// TIA Portal V16 export
// export: Created 2022-11-17T15:49:29.9822396Z, ExportSetting WithDefaults, DisplayName Totally Integrated Automation Portal, DisplayVersion V16 Update 6, DisplayName TIA Portal Version Control Interface, DisplayVersion V16 Update 2, DisplayName TIA Portal Openness, DisplayVersion V16 Update 6, DisplayName SINAMICS Startdrive Advanced, DisplayVersion V16 Update 5, DisplayName SINAMICS Startdrive G130, G150, S120, S150, SINAMICS MV, S210, DisplayVersion V16 Update 5, DisplayName SINAMICS Startdrive G110M, G120, G120C, G120D, G120P, G115D, DisplayVersion V16 Update 5, DisplayName STEP 7 Professional, DisplayVersion V16 Update 6, DisplayName STEP 7 Safety, DisplayVersion V16, DisplayName WinCC Advanced, DisplayVersion V16 Update 6
FUNCTION "FC86_Conveyor_5_IN_3_OUT" : Void   // FC86, LAD
TITLE = Conveyor_5_IN_3_OUT
{ S7_Optimized_Access := 'TRUE' }
VERSION : 0.1
// 5+3 (Fitembal)
// stored: AutoNumber false, IsIECCheckEnabled false, SetENOAutomatically false, UDAEnableTagReadback false
   VAR_TEMP   // added for the SCL form of the ladder/FBD networks
      _w1 : Bool;
      _w2 : Bool;
   END_VAR
BEGIN

REGION Network 1: Manual operation for conveyor
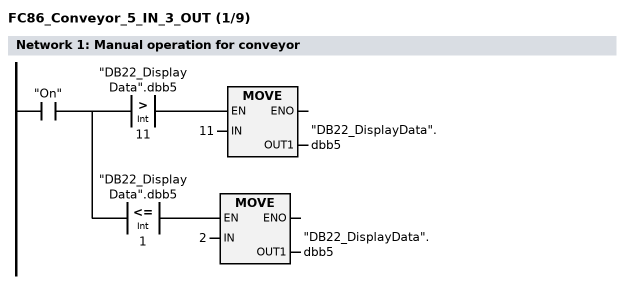
   RUNG wire#powerrail
      Contact( "On" )
      wire#w1
      { S7_Templates := "SrcType := Int" } GT_Contact(in1 := "DB22_DisplayData".dbb5, in2 := 11)
      { S7_GenerateENO := "TRUE" } Move(in := 11, out1 => "DB22_DisplayData".dbb5)
   END_RUNG
   RUNG wire#w1
      { S7_Templates := "SrcType := Int" } LE_Contact(in1 := "DB22_DisplayData".dbb5, in2 := 1)
      { S7_GenerateENO := "TRUE" } Move(in := 2, out1 => "DB22_DisplayData".dbb5)
   END_RUNG
   // the same network as SCL:
   IF "On" AND ("DB22_DisplayData".dbb5 > 11) THEN "DB22_DisplayData".dbb5 := 11; END_IF;
   IF "On" AND ("DB22_DisplayData".dbb5 <= 1) THEN "DB22_DisplayData".dbb5 := 2; END_IF;
END_REGION

REGION Network 2: Manual operation for conveyor
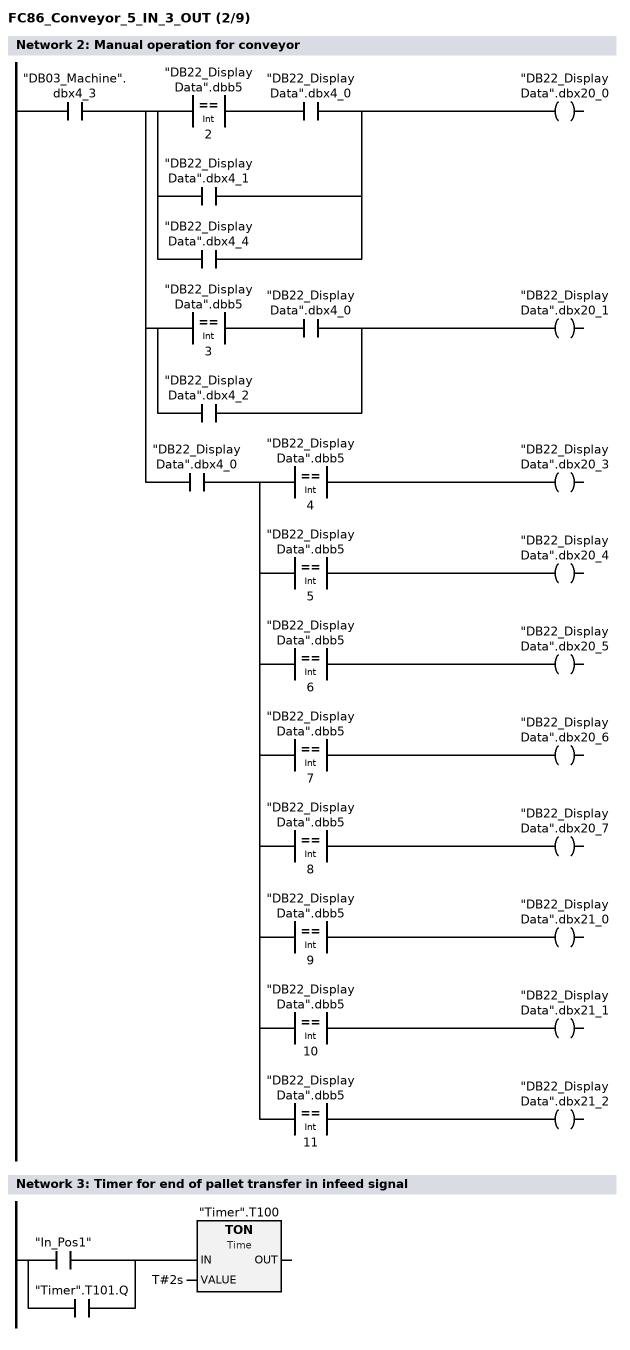
   RUNG wire#powerrail
      Contact( "DB03_Machine".dbx4_3 )
      wire#w1
      { S7_Templates := "SrcType := Int" } EQ_Contact(in1 := "DB22_DisplayData".dbb5, in2 := 2)
      Contact( "DB22_DisplayData".dbx4_0 )
      wire#w2
      Coil( "DB22_DisplayData".dbx20_0 )
   END_RUNG
   RUNG wire#w1
      Contact( "DB22_DisplayData".dbx4_1 )
   END_RUNG wire#w2
   RUNG wire#w1
      Contact( "DB22_DisplayData".dbx4_4 )
   END_RUNG wire#w2
   RUNG wire#w1
      { S7_Templates := "SrcType := Int" } EQ_Contact(in1 := "DB22_DisplayData".dbb5, in2 := 3)
      Contact( "DB22_DisplayData".dbx4_0 )
      wire#w3
      Coil( "DB22_DisplayData".dbx20_1 )
   END_RUNG
   RUNG wire#w1
      Contact( "DB22_DisplayData".dbx4_2 )
   END_RUNG wire#w3
   RUNG wire#w1
      Contact( "DB22_DisplayData".dbx4_0 )
      wire#w4
      { S7_Templates := "SrcType := Int" } EQ_Contact(in1 := "DB22_DisplayData".dbb5, in2 := 4)
      Coil( "DB22_DisplayData".dbx20_3 )
   END_RUNG
   RUNG wire#w4
      { S7_Templates := "SrcType := Int" } EQ_Contact(in1 := "DB22_DisplayData".dbb5, in2 := 5)
      Coil( "DB22_DisplayData".dbx20_4 )
   END_RUNG
   RUNG wire#w4
      { S7_Templates := "SrcType := Int" } EQ_Contact(in1 := "DB22_DisplayData".dbb5, in2 := 6)
      Coil( "DB22_DisplayData".dbx20_5 )
   END_RUNG
   RUNG wire#w4
      { S7_Templates := "SrcType := Int" } EQ_Contact(in1 := "DB22_DisplayData".dbb5, in2 := 7)
      Coil( "DB22_DisplayData".dbx20_6 )
   END_RUNG
   RUNG wire#w4
      { S7_Templates := "SrcType := Int" } EQ_Contact(in1 := "DB22_DisplayData".dbb5, in2 := 8)
      Coil( "DB22_DisplayData".dbx20_7 )
   END_RUNG
   RUNG wire#w4
      { S7_Templates := "SrcType := Int" } EQ_Contact(in1 := "DB22_DisplayData".dbb5, in2 := 9)
      Coil( "DB22_DisplayData".dbx21_0 )
   END_RUNG
   RUNG wire#w4
      { S7_Templates := "SrcType := Int" } EQ_Contact(in1 := "DB22_DisplayData".dbb5, in2 := 10)
      Coil( "DB22_DisplayData".dbx21_1 )
   END_RUNG
   RUNG wire#w4
      { S7_Templates := "SrcType := Int" } EQ_Contact(in1 := "DB22_DisplayData".dbb5, in2 := 11)
      Coil( "DB22_DisplayData".dbx21_2 )
   END_RUNG
   // the same network as SCL:
   "DB22_DisplayData".dbx20_0 := "DB03_Machine".dbx4_3 AND ((("DB22_DisplayData".dbb5 = 2) AND "DB22_DisplayData".dbx4_0) OR "DB22_DisplayData".dbx4_1 OR "DB22_DisplayData".dbx4_4);
   "DB22_DisplayData".dbx20_1 := "DB03_Machine".dbx4_3 AND ((("DB22_DisplayData".dbb5 = 3) AND "DB22_DisplayData".dbx4_0) OR "DB22_DisplayData".dbx4_2);
   #_w1 := "DB03_Machine".dbx4_3 AND "DB22_DisplayData".dbx4_0;
   "DB22_DisplayData".dbx20_3 := #_w1 AND ("DB22_DisplayData".dbb5 = 4);
   "DB22_DisplayData".dbx20_4 := #_w1 AND ("DB22_DisplayData".dbb5 = 5);
   "DB22_DisplayData".dbx20_5 := #_w1 AND ("DB22_DisplayData".dbb5 = 6);
   "DB22_DisplayData".dbx20_6 := #_w1 AND ("DB22_DisplayData".dbb5 = 7);
   "DB22_DisplayData".dbx20_7 := #_w1 AND ("DB22_DisplayData".dbb5 = 8);
   "DB22_DisplayData".dbx21_0 := #_w1 AND ("DB22_DisplayData".dbb5 = 9);
   "DB22_DisplayData".dbx21_1 := #_w1 AND ("DB22_DisplayData".dbb5 = 10);
   "DB22_DisplayData".dbx21_2 := #_w1 AND ("DB22_DisplayData".dbb5 = 11);
END_REGION

REGION Network 3: Timer for end of pallet transfer in infeed signal
   "Timer".T100.TON(IN := "In_Pos1" OR "Timer".T101.Q, PT := T#2s);   // TON coil
END_REGION

REGION Network 4: Timeout for conveyor pos1
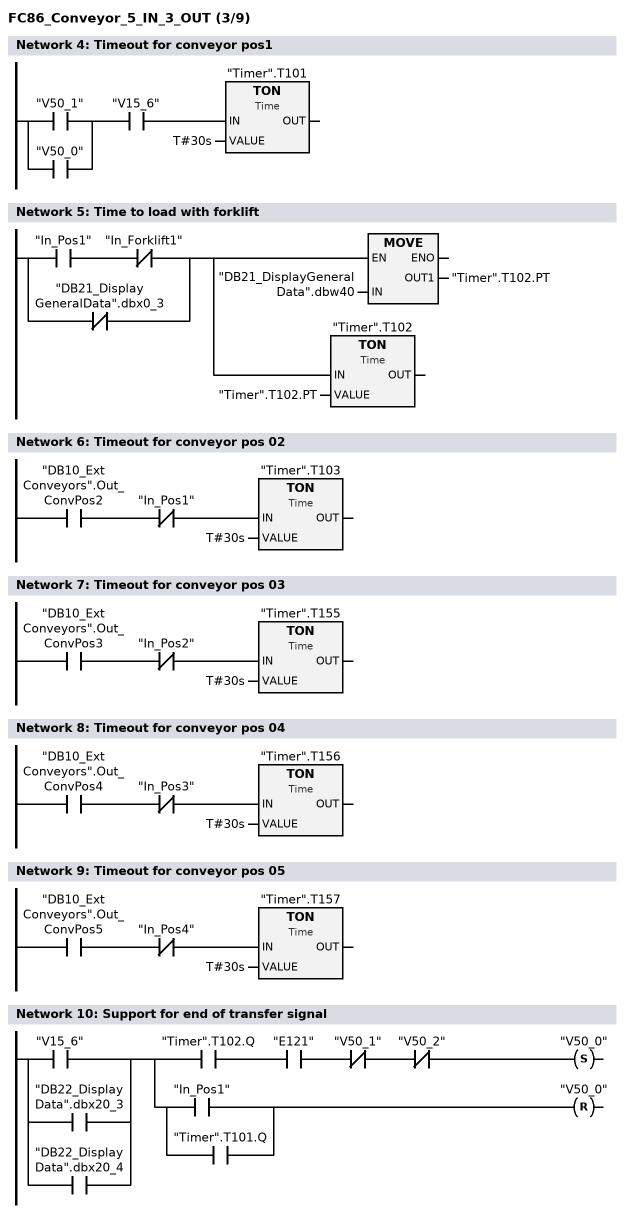
   "Timer".T101.TON(IN := ("V50_1" OR "V50_0") AND "V15_6", PT := T#30s);   // TON coil
END_REGION

REGION Network 5: Time to load with forklift
   #_w1 := ("In_Pos1" AND NOT "In_Forklift1") OR NOT "DB21_DisplayGeneralData".dbx0_3;
   IF #_w1 THEN "Timer".T102.PT := "DB21_DisplayGeneralData".dbw40; END_IF;
   "Timer".T102.TON(IN := #_w1, PT := "Timer".T102.PT);   // TON coil
END_REGION

REGION Network 6: Timeout for conveyor pos 02
   "Timer".T103.TON(IN := "DB10_ExtConveyors".Out_ConvPos2 AND NOT "In_Pos1", PT := T#30s);   // TON coil
END_REGION

REGION Network 7: Timeout for conveyor pos 03
   "Timer".T155.TON(IN := "DB10_ExtConveyors".Out_ConvPos3 AND NOT "In_Pos2", PT := T#30s);   // TON coil
END_REGION

REGION Network 8: Timeout for conveyor pos 04
   "Timer".T156.TON(IN := "DB10_ExtConveyors".Out_ConvPos4 AND NOT "In_Pos3", PT := T#30s);   // TON coil
END_REGION

REGION Network 9: Timeout for conveyor pos 05
   "Timer".T157.TON(IN := "DB10_ExtConveyors".Out_ConvPos5 AND NOT "In_Pos4", PT := T#30s);   // TON coil
END_REGION

REGION Network 10: Support for end of transfer signal
   RUNG wire#powerrail
      Contact( "V15_6" )
      wire#w1
      Contact( "Timer".T102.Q )
      Contact( "E121" )
      I_Contact( "V50_1" )
      I_Contact( "V50_2" )
      S_Coil( "V50_0" )
   END_RUNG
   RUNG wire#powerrail
      Contact( "DB22_DisplayData".dbx20_3 )
   END_RUNG wire#w1
   RUNG wire#powerrail
      Contact( "DB22_DisplayData".dbx20_4 )
   END_RUNG wire#w1
   RUNG wire#w1
      Contact( "In_Pos1" )
      wire#w2
      R_Coil( "V50_0" )
   END_RUNG
   RUNG wire#w1
      Contact( "Timer".T101.Q )
   END_RUNG wire#w2
   // the same network as SCL:
   #_w1 := "V15_6" OR "DB22_DisplayData".dbx20_3 OR "DB22_DisplayData".dbx20_4;
   IF #_w1 AND "Timer".T102.Q AND "E121" AND NOT "V50_1" AND NOT "V50_2" THEN "V50_0" := TRUE; END_IF;
   IF #_w1 AND ("In_Pos1" OR "Timer".T101.Q) THEN "V50_0" := FALSE; END_IF;
END_REGION

REGION Network 11: Transit memory for conveyor pos1
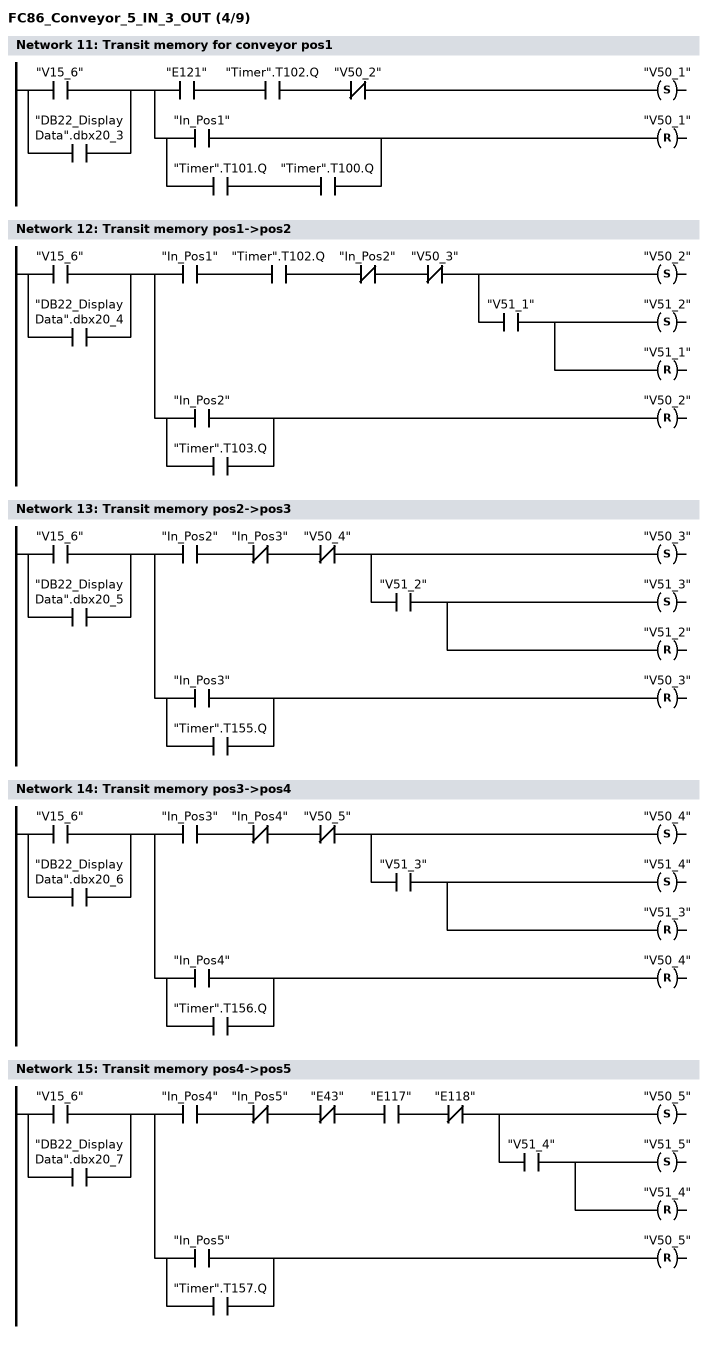
   RUNG wire#powerrail
      Contact( "V15_6" )
      wire#w1
      Contact( "E121" )
      Contact( "Timer".T102.Q )
      I_Contact( "V50_2" )
      S_Coil( "V50_1" )
   END_RUNG
   RUNG wire#powerrail
      Contact( "DB22_DisplayData".dbx20_3 )
   END_RUNG wire#w1
   RUNG wire#w1
      Contact( "In_Pos1" )
      wire#w2
      R_Coil( "V50_1" )
   END_RUNG
   RUNG wire#w1
      Contact( "Timer".T101.Q )
      Contact( "Timer".T100.Q )
   END_RUNG wire#w2
   // the same network as SCL:
   #_w1 := "V15_6" OR "DB22_DisplayData".dbx20_3;
   IF #_w1 AND "E121" AND "Timer".T102.Q AND NOT "V50_2" THEN "V50_1" := TRUE; END_IF;
   IF #_w1 AND ("In_Pos1" OR ("Timer".T101.Q AND "Timer".T100.Q)) THEN "V50_1" := FALSE; END_IF;
END_REGION

REGION Network 12: Transit memory pos1->pos2
   RUNG wire#powerrail
      Contact( "V15_6" )
      wire#w1
      Contact( "In_Pos1" )
      Contact( "Timer".T102.Q )
      I_Contact( "In_Pos2" )
      I_Contact( "V50_3" )
      wire#w2
      S_Coil( "V50_2" )
   END_RUNG
   RUNG wire#powerrail
      Contact( "DB22_DisplayData".dbx20_4 )
   END_RUNG wire#w1
   RUNG wire#w2
      Contact( "V51_1" )
      wire#w3
      S_Coil( "V51_2" )
   END_RUNG
   RUNG wire#w3
      R_Coil( "V51_1" )
   END_RUNG
   RUNG wire#w1
      Contact( "In_Pos2" )
      wire#w4
      R_Coil( "V50_2" )
   END_RUNG
   RUNG wire#w1
      Contact( "Timer".T103.Q )
   END_RUNG wire#w4
   // the same network as SCL:
   #_w1 := "V15_6" OR "DB22_DisplayData".dbx20_4;
   #_w2 := #_w1 AND "In_Pos1" AND "Timer".T102.Q AND NOT "In_Pos2" AND NOT "V50_3";
   IF #_w2 THEN "V50_2" := TRUE; END_IF;
   IF #_w2 AND "V51_1" THEN
       "V51_2" := TRUE;
       "V51_1" := FALSE;
   END_IF;
   IF #_w1 AND ("In_Pos2" OR "Timer".T103.Q) THEN "V50_2" := FALSE; END_IF;
END_REGION

REGION Network 13: Transit memory pos2->pos3
   RUNG wire#powerrail
      Contact( "V15_6" )
      wire#w1
      Contact( "In_Pos2" )
      I_Contact( "In_Pos3" )
      I_Contact( "V50_4" )
      wire#w2
      S_Coil( "V50_3" )
   END_RUNG
   RUNG wire#powerrail
      Contact( "DB22_DisplayData".dbx20_5 )
   END_RUNG wire#w1
   RUNG wire#w2
      Contact( "V51_2" )
      wire#w3
      S_Coil( "V51_3" )
   END_RUNG
   RUNG wire#w3
      R_Coil( "V51_2" )
   END_RUNG
   RUNG wire#w1
      Contact( "In_Pos3" )
      wire#w4
      R_Coil( "V50_3" )
   END_RUNG
   RUNG wire#w1
      Contact( "Timer".T155.Q )
   END_RUNG wire#w4
   // the same network as SCL:
   #_w1 := "V15_6" OR "DB22_DisplayData".dbx20_5;
   #_w2 := #_w1 AND "In_Pos2" AND NOT "In_Pos3" AND NOT "V50_4";
   IF #_w2 THEN "V50_3" := TRUE; END_IF;
   IF #_w2 AND "V51_2" THEN
       "V51_3" := TRUE;
       "V51_2" := FALSE;
   END_IF;
   IF #_w1 AND ("In_Pos3" OR "Timer".T155.Q) THEN "V50_3" := FALSE; END_IF;
END_REGION

REGION Network 14: Transit memory pos3->pos4
   RUNG wire#powerrail
      Contact( "V15_6" )
      wire#w1
      Contact( "In_Pos3" )
      I_Contact( "In_Pos4" )
      I_Contact( "V50_5" )
      wire#w2
      S_Coil( "V50_4" )
   END_RUNG
   RUNG wire#powerrail
      Contact( "DB22_DisplayData".dbx20_6 )
   END_RUNG wire#w1
   RUNG wire#w2
      Contact( "V51_3" )
      wire#w3
      S_Coil( "V51_4" )
   END_RUNG
   RUNG wire#w3
      R_Coil( "V51_3" )
   END_RUNG
   RUNG wire#w1
      Contact( "In_Pos4" )
      wire#w4
      R_Coil( "V50_4" )
   END_RUNG
   RUNG wire#w1
      Contact( "Timer".T156.Q )
   END_RUNG wire#w4
   // the same network as SCL:
   #_w1 := "V15_6" OR "DB22_DisplayData".dbx20_6;
   #_w2 := #_w1 AND "In_Pos3" AND NOT "In_Pos4" AND NOT "V50_5";
   IF #_w2 THEN "V50_4" := TRUE; END_IF;
   IF #_w2 AND "V51_3" THEN
       "V51_4" := TRUE;
       "V51_3" := FALSE;
   END_IF;
   IF #_w1 AND ("In_Pos4" OR "Timer".T156.Q) THEN "V50_4" := FALSE; END_IF;
END_REGION

REGION Network 15: Transit memory pos4->pos5
   RUNG wire#powerrail
      Contact( "V15_6" )
      wire#w1
      Contact( "In_Pos4" )
      I_Contact( "In_Pos5" )
      I_Contact( "E43" )
      Contact( "E117" )
      I_Contact( "E118" )
      wire#w2
      S_Coil( "V50_5" )
   END_RUNG
   RUNG wire#powerrail
      Contact( "DB22_DisplayData".dbx20_7 )
   END_RUNG wire#w1
   RUNG wire#w2
      Contact( "V51_4" )
      wire#w3
      S_Coil( "V51_5" )
   END_RUNG
   RUNG wire#w3
      R_Coil( "V51_4" )
   END_RUNG
   RUNG wire#w1
      Contact( "In_Pos5" )
      wire#w4
      R_Coil( "V50_5" )
   END_RUNG
   RUNG wire#w1
      Contact( "Timer".T157.Q )
   END_RUNG wire#w4
   // the same network as SCL:
   #_w1 := "V15_6" OR "DB22_DisplayData".dbx20_7;
   #_w2 := #_w1 AND "In_Pos4" AND NOT "In_Pos5" AND NOT "E43" AND "E117" AND NOT "E118";
   IF #_w2 THEN "V50_5" := TRUE; END_IF;
   IF #_w2 AND "V51_4" THEN
       "V51_5" := TRUE;
       "V51_4" := FALSE;
   END_IF;
   IF #_w1 AND ("In_Pos5" OR "Timer".T157.Q) THEN "V50_5" := FALSE; END_IF;
END_REGION

REGION Network 16: Ready to receive pallet in infeed signal
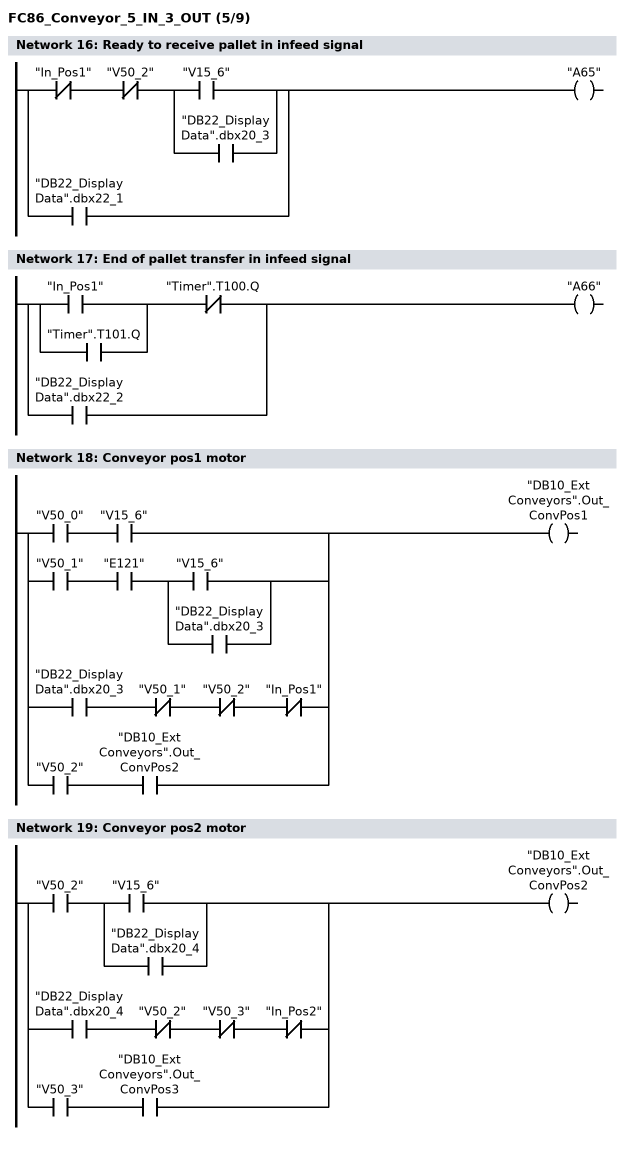
   RUNG wire#powerrail
      I_Contact( "In_Pos1" )
      I_Contact( "V50_2" )
      wire#w1
      Contact( "V15_6" )
      wire#w2
      Coil( "A65" )
   END_RUNG
   RUNG wire#w1
      Contact( "DB22_DisplayData".dbx20_3 )
   END_RUNG wire#w2
   RUNG wire#powerrail
      Contact( "DB22_DisplayData".dbx22_1 )
   END_RUNG wire#w2
   // the same network as SCL:
   "A65" := (NOT "In_Pos1" AND NOT "V50_2" AND ("V15_6" OR "DB22_DisplayData".dbx20_3)) OR "DB22_DisplayData".dbx22_1;
END_REGION

REGION Network 17: End of pallet transfer in infeed signal
   RUNG wire#powerrail
      Contact( "In_Pos1" )
      wire#w1
      I_Contact( "Timer".T100.Q )
      wire#w2
      Coil( "A66" )
   END_RUNG
   RUNG wire#powerrail
      Contact( "Timer".T101.Q )
   END_RUNG wire#w1
   RUNG wire#powerrail
      Contact( "DB22_DisplayData".dbx22_2 )
   END_RUNG wire#w2
   // the same network as SCL:
   "A66" := (("In_Pos1" OR "Timer".T101.Q) AND NOT "Timer".T100.Q) OR "DB22_DisplayData".dbx22_2;
END_REGION

REGION Network 18: Conveyor pos1 motor
   RUNG wire#powerrail
      Contact( "V50_0" )
      Contact( "V15_6" )
      wire#w1
      Coil( "DB10_ExtConveyors".Out_ConvPos1 )
   END_RUNG
   RUNG wire#powerrail
      Contact( "V50_1" )
      Contact( "E121" )
      wire#w2
      Contact( "V15_6" )
   END_RUNG wire#w1
   RUNG wire#w2
      Contact( "DB22_DisplayData".dbx20_3 )
   END_RUNG wire#w1
   RUNG wire#powerrail
      Contact( "DB22_DisplayData".dbx20_3 )
      I_Contact( "V50_1" )
      I_Contact( "V50_2" )
      I_Contact( "In_Pos1" )
   END_RUNG wire#w1
   RUNG wire#powerrail
      Contact( "V50_2" )
      Contact( "DB10_ExtConveyors".Out_ConvPos2 )
   END_RUNG wire#w1
   // the same network as SCL:
   "DB10_ExtConveyors".Out_ConvPos1 := ("V50_0" AND "V15_6") OR ("V50_1" AND "E121" AND ("V15_6" OR "DB22_DisplayData".dbx20_3)) OR ("DB22_DisplayData".dbx20_3 AND NOT "V50_1" AND NOT "V50_2" AND NOT "In_Pos1") OR ("V50_2" AND "DB10_ExtConveyors".Out_ConvPos2);
END_REGION

REGION Network 19: Conveyor pos2 motor
   RUNG wire#powerrail
      Contact( "V50_2" )
      wire#w1
      Contact( "V15_6" )
      wire#w2
      Coil( "DB10_ExtConveyors".Out_ConvPos2 )
   END_RUNG
   RUNG wire#w1
      Contact( "DB22_DisplayData".dbx20_4 )
   END_RUNG wire#w2
   RUNG wire#powerrail
      Contact( "DB22_DisplayData".dbx20_4 )
      I_Contact( "V50_2" )
      I_Contact( "V50_3" )
      I_Contact( "In_Pos2" )
   END_RUNG wire#w2
   RUNG wire#powerrail
      Contact( "V50_3" )
      Contact( "DB10_ExtConveyors".Out_ConvPos3 )
   END_RUNG wire#w2
   // the same network as SCL:
   "DB10_ExtConveyors".Out_ConvPos2 := ("V50_2" AND ("V15_6" OR "DB22_DisplayData".dbx20_4)) OR ("DB22_DisplayData".dbx20_4 AND NOT "V50_2" AND NOT "V50_3" AND NOT "In_Pos2") OR ("V50_3" AND "DB10_ExtConveyors".Out_ConvPos3);
END_REGION

REGION Network 20: Conveyor pos3 motor
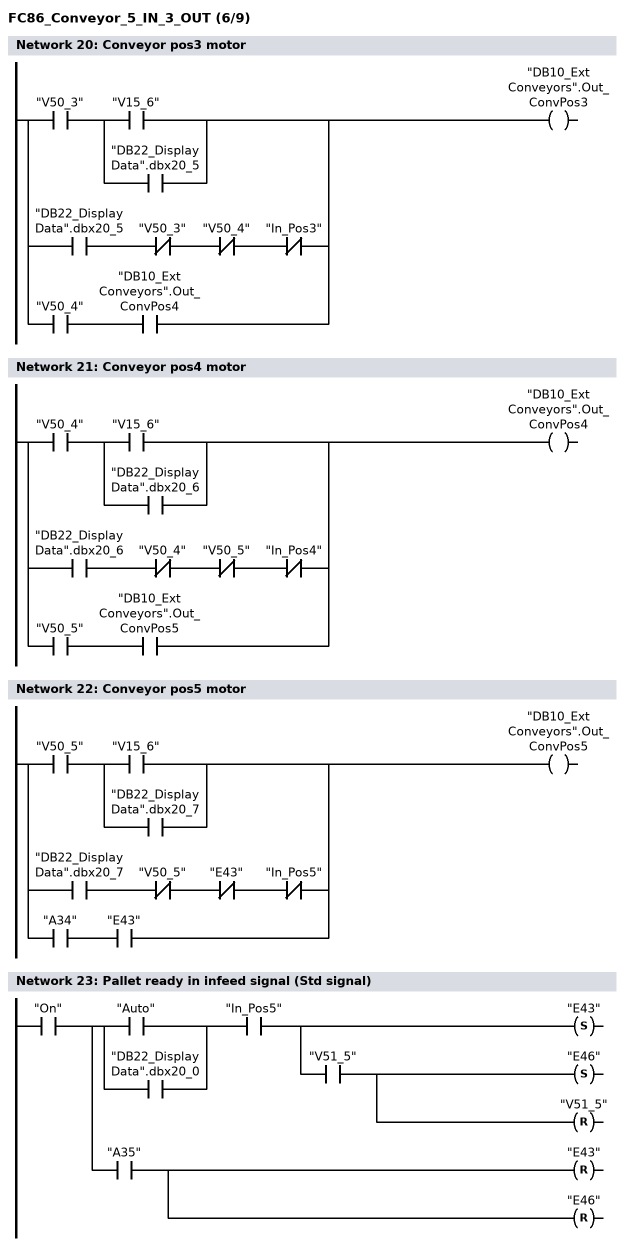
   RUNG wire#powerrail
      Contact( "V50_3" )
      wire#w1
      Contact( "V15_6" )
      wire#w2
      Coil( "DB10_ExtConveyors".Out_ConvPos3 )
   END_RUNG
   RUNG wire#w1
      Contact( "DB22_DisplayData".dbx20_5 )
   END_RUNG wire#w2
   RUNG wire#powerrail
      Contact( "DB22_DisplayData".dbx20_5 )
      I_Contact( "V50_3" )
      I_Contact( "V50_4" )
      I_Contact( "In_Pos3" )
   END_RUNG wire#w2
   RUNG wire#powerrail
      Contact( "V50_4" )
      Contact( "DB10_ExtConveyors".Out_ConvPos4 )
   END_RUNG wire#w2
   // the same network as SCL:
   "DB10_ExtConveyors".Out_ConvPos3 := ("V50_3" AND ("V15_6" OR "DB22_DisplayData".dbx20_5)) OR ("DB22_DisplayData".dbx20_5 AND NOT "V50_3" AND NOT "V50_4" AND NOT "In_Pos3") OR ("V50_4" AND "DB10_ExtConveyors".Out_ConvPos4);
END_REGION

REGION Network 21: Conveyor pos4 motor
   RUNG wire#powerrail
      Contact( "V50_4" )
      wire#w1
      Contact( "V15_6" )
      wire#w2
      Coil( "DB10_ExtConveyors".Out_ConvPos4 )
   END_RUNG
   RUNG wire#w1
      Contact( "DB22_DisplayData".dbx20_6 )
   END_RUNG wire#w2
   RUNG wire#powerrail
      Contact( "DB22_DisplayData".dbx20_6 )
      I_Contact( "V50_4" )
      I_Contact( "V50_5" )
      I_Contact( "In_Pos4" )
   END_RUNG wire#w2
   RUNG wire#powerrail
      Contact( "V50_5" )
      Contact( "DB10_ExtConveyors".Out_ConvPos5 )
   END_RUNG wire#w2
   // the same network as SCL:
   "DB10_ExtConveyors".Out_ConvPos4 := ("V50_4" AND ("V15_6" OR "DB22_DisplayData".dbx20_6)) OR ("DB22_DisplayData".dbx20_6 AND NOT "V50_4" AND NOT "V50_5" AND NOT "In_Pos4") OR ("V50_5" AND "DB10_ExtConveyors".Out_ConvPos5);
END_REGION

REGION Network 22: Conveyor pos5 motor
   RUNG wire#powerrail
      Contact( "V50_5" )
      wire#w1
      Contact( "V15_6" )
      wire#w2
      Coil( "DB10_ExtConveyors".Out_ConvPos5 )
   END_RUNG
   RUNG wire#w1
      Contact( "DB22_DisplayData".dbx20_7 )
   END_RUNG wire#w2
   RUNG wire#powerrail
      Contact( "DB22_DisplayData".dbx20_7 )
      I_Contact( "V50_5" )
      I_Contact( "E43" )
      I_Contact( "In_Pos5" )
   END_RUNG wire#w2
   RUNG wire#powerrail
      Contact( "A34" )
      Contact( "E43" )
   END_RUNG wire#w2
   // the same network as SCL:
   "DB10_ExtConveyors".Out_ConvPos5 := ("V50_5" AND ("V15_6" OR "DB22_DisplayData".dbx20_7)) OR ("DB22_DisplayData".dbx20_7 AND NOT "V50_5" AND NOT "E43" AND NOT "In_Pos5") OR ("A34" AND "E43");
END_REGION

REGION Network 23: Pallet ready in infeed signal (Std signal)
   RUNG wire#powerrail
      Contact( "On" )
      wire#w1
      Contact( "Auto" )
      wire#w2
      Contact( "In_Pos5" )
      wire#w3
      S_Coil( "E43" )
   END_RUNG
   RUNG wire#w1
      Contact( "DB22_DisplayData".dbx20_0 )
   END_RUNG wire#w2
   RUNG wire#w3
      Contact( "V51_5" )
      wire#w4
      S_Coil( "E46" )
   END_RUNG
   RUNG wire#w4
      R_Coil( "V51_5" )
   END_RUNG
   RUNG wire#w1
      Contact( "A35" )
      wire#w5
      R_Coil( "E43" )
   END_RUNG
   RUNG wire#w5
      R_Coil( "E46" )
   END_RUNG
   // the same network as SCL:
   #_w1 := "On" AND ("Auto" OR "DB22_DisplayData".dbx20_0) AND "In_Pos5";
   IF #_w1 THEN "E43" := TRUE; END_IF;
   IF #_w1 AND "V51_5" THEN
       "E46" := TRUE;
       "V51_5" := FALSE;
   END_IF;
   IF "On" AND "A35" THEN
       "E43" := FALSE;
       "E46" := FALSE;
   END_IF;
END_REGION

REGION Network 24: Memory to exclude wrapping in pos 1
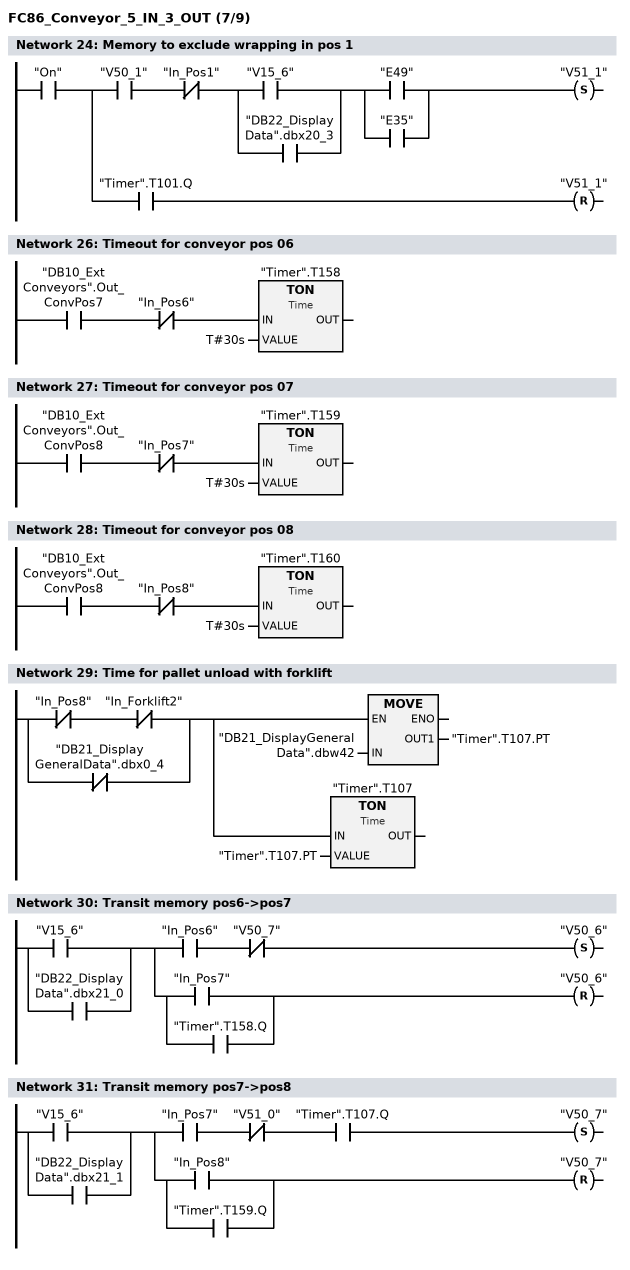
   RUNG wire#powerrail
      Contact( "On" )
      wire#w1
      Contact( "V50_1" )
      I_Contact( "In_Pos1" )
      wire#w2
      Contact( "V15_6" )
      wire#w3
      Contact( "E49" )
      wire#w4
      S_Coil( "V51_1" )
   END_RUNG
   RUNG wire#w2
      Contact( "DB22_DisplayData".dbx20_3 )
   END_RUNG wire#w3
   RUNG wire#w3
      Contact( "E35" )
   END_RUNG wire#w4
   RUNG wire#w1
      Contact( "Timer".T101.Q )
      R_Coil( "V51_1" )
   END_RUNG
   // the same network as SCL:
   IF "On" AND "V50_1" AND NOT "In_Pos1" AND ("V15_6" OR "DB22_DisplayData".dbx20_3) AND ("E49" OR "E35") THEN
       "V51_1" := TRUE;
   END_IF;
   IF "On" AND "Timer".T101.Q THEN "V51_1" := FALSE; END_IF;
END_REGION

REGION Network 25: >>>>>>> OUTFEED CONVEYOR <<<<<<<<
END_REGION

REGION Network 26: Timeout for conveyor pos 06
   "Timer".T158.TON(IN := "DB10_ExtConveyors".Out_ConvPos7 AND NOT "In_Pos6", PT := T#30s);   // TON coil
END_REGION

REGION Network 27: Timeout for conveyor pos 07
   "Timer".T159.TON(IN := "DB10_ExtConveyors".Out_ConvPos8 AND NOT "In_Pos7", PT := T#30s);   // TON coil
END_REGION

REGION Network 28: Timeout for conveyor pos 08
   "Timer".T160.TON(IN := "DB10_ExtConveyors".Out_ConvPos8 AND NOT "In_Pos8", PT := T#30s);   // TON coil
END_REGION

REGION Network 29: Time for pallet unload with forklift
   #_w1 := (NOT "In_Pos8" AND NOT "In_Forklift2") OR NOT "DB21_DisplayGeneralData".dbx0_4;
   IF #_w1 THEN "Timer".T107.PT := "DB21_DisplayGeneralData".dbw42; END_IF;
   "Timer".T107.TON(IN := #_w1, PT := "Timer".T107.PT);   // TON coil
END_REGION

REGION Network 30: Transit memory pos6->pos7
   RUNG wire#powerrail
      Contact( "V15_6" )
      wire#w1
      Contact( "In_Pos6" )
      I_Contact( "V50_7" )
      S_Coil( "V50_6" )
   END_RUNG
   RUNG wire#powerrail
      Contact( "DB22_DisplayData".dbx21_0 )
   END_RUNG wire#w1
   RUNG wire#w1
      Contact( "In_Pos7" )
      wire#w2
      R_Coil( "V50_6" )
   END_RUNG
   RUNG wire#w1
      Contact( "Timer".T158.Q )
   END_RUNG wire#w2
   // the same network as SCL:
   #_w1 := "V15_6" OR "DB22_DisplayData".dbx21_0;
   IF #_w1 AND "In_Pos6" AND NOT "V50_7" THEN "V50_6" := TRUE; END_IF;
   IF #_w1 AND ("In_Pos7" OR "Timer".T158.Q) THEN "V50_6" := FALSE; END_IF;
END_REGION

REGION Network 31: Transit memory pos7->pos8
   RUNG wire#powerrail
      Contact( "V15_6" )
      wire#w1
      Contact( "In_Pos7" )
      I_Contact( "V51_0" )
      Contact( "Timer".T107.Q )
      S_Coil( "V50_7" )
   END_RUNG
   RUNG wire#powerrail
      Contact( "DB22_DisplayData".dbx21_1 )
   END_RUNG wire#w1
   RUNG wire#w1
      Contact( "In_Pos8" )
      wire#w2
      R_Coil( "V50_7" )
   END_RUNG
   RUNG wire#w1
      Contact( "Timer".T159.Q )
   END_RUNG wire#w2
   // the same network as SCL:
   #_w1 := "V15_6" OR "DB22_DisplayData".dbx21_1;
   IF #_w1 AND "In_Pos7" AND NOT "V51_0" AND "Timer".T107.Q THEN "V50_7" := TRUE; END_IF;
   IF #_w1 AND ("In_Pos8" OR "Timer".T159.Q) THEN "V50_7" := FALSE; END_IF;
END_REGION

REGION Network 32: Outfeed conveyor pos.8 unload
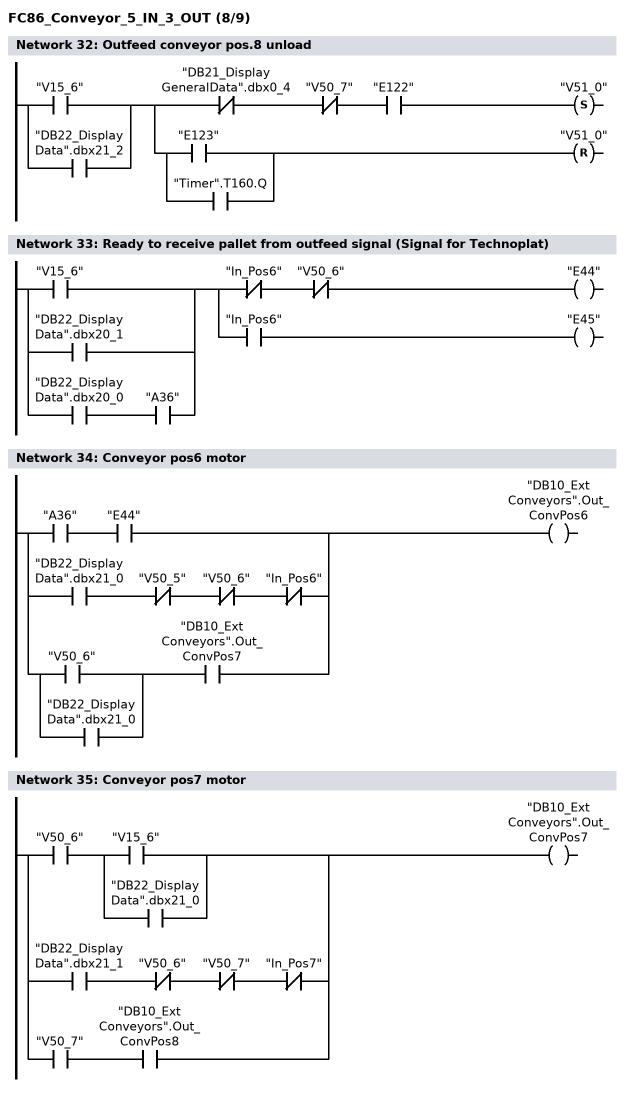
   RUNG wire#powerrail
      Contact( "V15_6" )
      wire#w1
      I_Contact( "DB21_DisplayGeneralData".dbx0_4 )
      I_Contact( "V50_7" )
      Contact( "E122" )
      S_Coil( "V51_0" )
   END_RUNG
   RUNG wire#powerrail
      Contact( "DB22_DisplayData".dbx21_2 )
   END_RUNG wire#w1
   RUNG wire#w1
      Contact( "E123" )
      wire#w2
      R_Coil( "V51_0" )
   END_RUNG
   RUNG wire#w1
      Contact( "Timer".T160.Q )
   END_RUNG wire#w2
   // the same network as SCL:
   #_w1 := "V15_6" OR "DB22_DisplayData".dbx21_2;
   IF #_w1 AND NOT "DB21_DisplayGeneralData".dbx0_4 AND NOT "V50_7" AND "E122" THEN "V51_0" := TRUE; END_IF;
   IF #_w1 AND ("E123" OR "Timer".T160.Q) THEN "V51_0" := FALSE; END_IF;
END_REGION

REGION Network 33: Ready to receive pallet from outfeed signal (Signal for Technoplat)
   RUNG wire#powerrail
      Contact( "V15_6" )
      wire#w1
      I_Contact( "In_Pos6" )
      I_Contact( "V50_6" )
      Coil( "E44" )
   END_RUNG
   RUNG wire#powerrail
      Contact( "DB22_DisplayData".dbx20_1 )
   END_RUNG wire#w1
   RUNG wire#powerrail
      Contact( "DB22_DisplayData".dbx20_0 )
      Contact( "A36" )
   END_RUNG wire#w1
   RUNG wire#w1
      Contact( "In_Pos6" )
      Coil( "E45" )
   END_RUNG
   // the same network as SCL:
   #_w1 := "V15_6" OR "DB22_DisplayData".dbx20_1 OR ("DB22_DisplayData".dbx20_0 AND "A36");
   "E44" := #_w1 AND NOT "In_Pos6" AND NOT "V50_6";
   "E45" := #_w1 AND "In_Pos6";
END_REGION

REGION Network 34: Conveyor pos6 motor
   RUNG wire#powerrail
      Contact( "A36" )
      Contact( "E44" )
      wire#w1
      Coil( "DB10_ExtConveyors".Out_ConvPos6 )
   END_RUNG
   RUNG wire#powerrail
      Contact( "DB22_DisplayData".dbx21_0 )
      I_Contact( "V50_5" )
      I_Contact( "V50_6" )
      I_Contact( "In_Pos6" )
   END_RUNG wire#w1
   RUNG wire#powerrail
      Contact( "V50_6" )
      wire#w2
      Contact( "DB10_ExtConveyors".Out_ConvPos7 )
   END_RUNG wire#w1
   RUNG wire#powerrail
      Contact( "DB22_DisplayData".dbx21_0 )
   END_RUNG wire#w2
   // the same network as SCL:
   "DB10_ExtConveyors".Out_ConvPos6 := ("A36" AND "E44") OR ("DB22_DisplayData".dbx21_0 AND NOT "V50_5" AND NOT "V50_6" AND NOT "In_Pos6") OR (("V50_6" OR "DB22_DisplayData".dbx21_0) AND "DB10_ExtConveyors".Out_ConvPos7);
END_REGION

REGION Network 35: Conveyor pos7 motor
   RUNG wire#powerrail
      Contact( "V50_6" )
      wire#w1
      Contact( "V15_6" )
      wire#w2
      Coil( "DB10_ExtConveyors".Out_ConvPos7 )
   END_RUNG
   RUNG wire#w1
      Contact( "DB22_DisplayData".dbx21_0 )
   END_RUNG wire#w2
   RUNG wire#powerrail
      Contact( "DB22_DisplayData".dbx21_1 )
      I_Contact( "V50_6" )
      I_Contact( "V50_7" )
      I_Contact( "In_Pos7" )
   END_RUNG wire#w2
   RUNG wire#powerrail
      Contact( "V50_7" )
      Contact( "DB10_ExtConveyors".Out_ConvPos8 )
   END_RUNG wire#w2
   // the same network as SCL:
   "DB10_ExtConveyors".Out_ConvPos7 := ("V50_6" AND ("V15_6" OR "DB22_DisplayData".dbx21_0)) OR ("DB22_DisplayData".dbx21_1 AND NOT "V50_6" AND NOT "V50_7" AND NOT "In_Pos7") OR ("V50_7" AND "DB10_ExtConveyors".Out_ConvPos8);
END_REGION

REGION Network 36: Conveyor pos8 motor
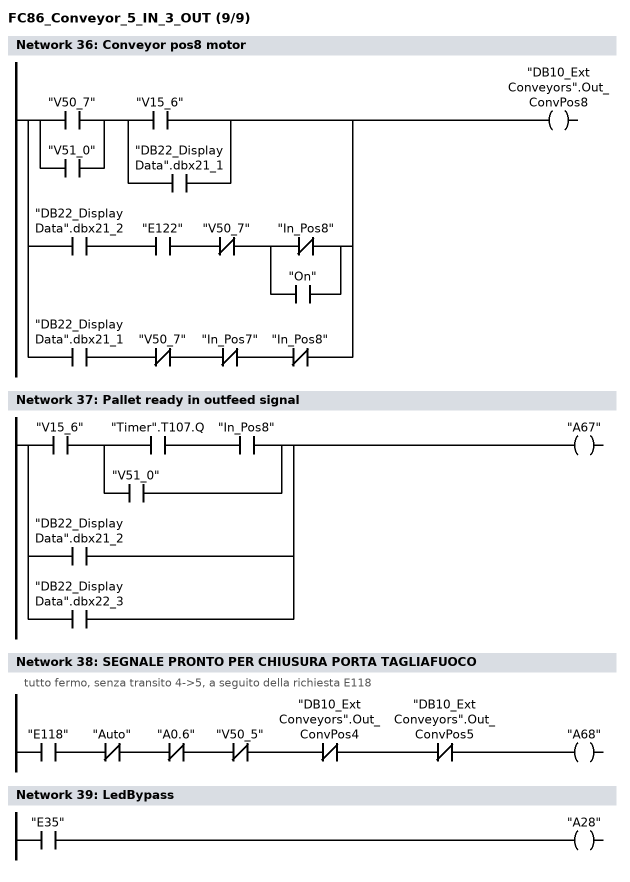
   RUNG wire#powerrail
      Contact( "V50_7" )
      wire#w1
      Contact( "V15_6" )
      wire#w2
      Coil( "DB10_ExtConveyors".Out_ConvPos8 )
   END_RUNG
   RUNG wire#powerrail
      Contact( "V51_0" )
   END_RUNG wire#w1
   RUNG wire#w1
      Contact( "DB22_DisplayData".dbx21_1 )
   END_RUNG wire#w2
   RUNG wire#powerrail
      Contact( "DB22_DisplayData".dbx21_2 )
      Contact( "E122" )
      I_Contact( "V50_7" )
      wire#w3
      I_Contact( "In_Pos8" )
   END_RUNG wire#w2
   RUNG wire#w3
      Contact( "On" )
   END_RUNG wire#w2
   RUNG wire#powerrail
      Contact( "DB22_DisplayData".dbx21_1 )
      I_Contact( "V50_7" )
      I_Contact( "In_Pos7" )
      I_Contact( "In_Pos8" )
   END_RUNG wire#w2
   // the same network as SCL:
   "DB10_ExtConveyors".Out_ConvPos8 := (("V50_7" OR "V51_0") AND ("V15_6" OR "DB22_DisplayData".dbx21_1)) OR ("DB22_DisplayData".dbx21_2 AND "E122" AND NOT "V50_7" AND (NOT "In_Pos8" OR "On")) OR ("DB22_DisplayData".dbx21_1 AND NOT "V50_7" AND NOT "In_Pos7" AND NOT "In_Pos8");
END_REGION

REGION Network 37: Pallet ready in outfeed signal
   RUNG wire#powerrail
      Contact( "V15_6" )
      wire#w1
      Contact( "Timer".T107.Q )
      Contact( "In_Pos8" )
      wire#w2
      Coil( "A67" )
   END_RUNG
   RUNG wire#w1
      Contact( "V51_0" )
   END_RUNG wire#w2
   RUNG wire#powerrail
      Contact( "DB22_DisplayData".dbx21_2 )
   END_RUNG wire#w2
   RUNG wire#powerrail
      Contact( "DB22_DisplayData".dbx22_3 )
   END_RUNG wire#w2
   // the same network as SCL:
   "A67" := ("V15_6" AND (("Timer".T107.Q AND "In_Pos8") OR "V51_0")) OR "DB22_DisplayData".dbx21_2 OR "DB22_DisplayData".dbx22_3;
END_REGION

REGION Network 38: SEGNALE PRONTO PER CHIUSURA PORTA TAGLIAFUOCO
   // tutto fermo, senza transito 4->5, a seguito della richiesta E118
   RUNG wire#powerrail
      Contact( "E118" )
      I_Contact( "Auto" )
      I_Contact( "A0.6" )
      I_Contact( "V50_5" )
      I_Contact( "DB10_ExtConveyors".Out_ConvPos4 )
      I_Contact( "DB10_ExtConveyors".Out_ConvPos5 )
      Coil( "A68" )
   END_RUNG
   // the same network as SCL:
   "A68" := "E118" AND NOT "Auto" AND NOT "A0.6" AND NOT "V50_5" AND NOT "DB10_ExtConveyors".Out_ConvPos4 AND NOT "DB10_ExtConveyors".Out_ConvPos5;
END_REGION

REGION Network 39: LedBypass
   RUNG wire#powerrail
      Contact( "E35" )
      Coil( "A28" )
   END_RUNG
   // the same network as SCL:
   "A28" := "E35";
END_REGION
END_FUNCTION
